Staubli VAL3: setAction.pgx

public program setAction(string& x_sAction[], num x_nIndex, bool x_bType)
  local string l_sInstruction
  local num i
begin
  // get the instruction and fill as an array
  if x_nIndex>=0
    if x_sAction[0]!="" or x_sAction[1]!="" or x_sAction[2]!=""
      // array to string
      l_sInstruction=x_sAction[0]
      for i=1 to size(x_sAction)-1
        l_sInstruction=l_sInstruction+"^"+x_sAction[i]
      endFor
    else
      // set empty
      l_sInstruction=""
    endIf
    // save the data
    if x_bType
      // take gun ON
      saveTool:sActionON[x_nIndex]=l_sInstruction
    else
      // take gun OFF
      saveTool:sActionOFF[x_nIndex]=l_sInstruction
    endIf
  endIf
end
